FUNCTION_BLOCK FB_ActorDownCommand IMPLEMENTS I_Command
VAR
	refFlyingHoist : REFERENCE TO FB_FlyingHoist;
END_VAR

METHOD Execute
IF (__ISVALIDREF(THIS^.refFlyingHoist)) THEN
	THIS^.refFlyingHoist.HoistEnable();
	THIS^.refFlyingHoist.ActorDown();
END_IF
END_METHOD

METHOD FB_init : BOOL
VAR_INPUT
	bInitRetains 	: BOOL; // if TRUE, the retain variables are initialized (warm start / cold start)
	bInCopyCode 	: BOOL;  // if TRUE, the instance afterwards gets moved into the copy code (online change)
	refFlyingHoist 	: REFERENCE TO FB_FlyingHoist;
END_VAR
IF (__ISVALIDREF(refFlyingHoist)) THEN
	THIS^.refFlyingHoist REF= refFlyingHoist;
ELSE
	THIS^.refFlyingHoist REF= 0;
END_IF
END_METHOD

END_FUNCTION_BLOCK

(* stored: Version 1.1.0.1, ProductVersion 3.1.4022.18
   POU FB_ActorDownCommand: Id {2078b464-5b40-44e8-8a80-8b442178bb99}, SpecialFunc None
   Method Execute: Id {c276a850-a646-4234-97a7-07704f73885f}
   Method FB_init: Id {920cab80-d358-41f7-9d8d-cb464ed6e5e5} *)
